// TIA Portal V19 export
DATA_BLOCK "PPrgArchive15"   // DB516
// stored: IsOnlyStoredInLoadMemory true, MemoryReserve 0, Namespace G
   VAR RETAIN
      PRG : Array[1401..1500] of "PPrg_Data";
   END_VAR
BEGIN
END_DATA_BLOCK
